TYPE U_Recived_bytes_from_Navitrol : UNION
		Header : ST_SupervisorHeader;
		Bytes  : ARRAY[0..5000] OF UINT;
	END_UNION
END_TYPE

(* stored: Version 1.1.0.1, ProductVersion 3.1.4026.17
   DUT U_Recived_bytes_from_Navitrol: Id {6436758d-6468-4e03-9bd1-aa20a5bb5423} *)
